// TwinCAT 3 PLC project WriteStringArrayToFile_Plc
// ProgramVersion: 3.1.4023.0
// libraries:
//   Tc2_Standard, * (Beckhoff Automation GmbH)
//   Tc2_System, * (Beckhoff Automation GmbH)
//   Tc3_Module, * (Beckhoff Automation GmbH)
// project tree:
//   / PlcTask.TcTTO
//   POUs/ FB_FillTestArray.TcPOU, FB_WriteStringArrayToFile.TcPOU, MAIN.TcPOU
// real-time tasks:
//   TASK PlcTask: cycle T#10ms, priority 20, ADS port 350

CONFIGURATION WriteStringArrayToFile_Plc
    RESOURCE PLC ON TwinCAT3
        TASK PlcTask(INTERVAL := T#10ms, PRIORITY := 20);
        PROGRAM MAIN WITH PlcTask : MAIN;
    END_RESOURCE
END_CONFIGURATION

// ---- POUs/MAIN.TcPOU
PROGRAM MAIN
VAR
	straTestStringArray	: ARRAY [1..10] OF STRING(255);
	fbFillArray	: FB_FillTestArray;
	fbWriteArray	: FB_WriteStringArrayToFile;
	
	bTestFillArray	: BOOL;
	bTestWriteArray	: BOOL;
	
	bTestOpen		: BOOL;
	bTestClose		: BOOL;
	
	fbFileOpen		: FB_FileOpen;
	fbFileClose		: FB_FileClose;
	
END_VAR

IF(_TaskInfo[GETCURTASKINDEXEX()].FirstCycle) THEN
	; // Do Nothing
END_IF


// Run the fill array FB 
fbFillArray(straArrayToFill	:= straTestStringArray);

// Run the file write array
fbWriteArray(straArrayToWrite	:= straTestStringArray);

IF(bTestFillArray) THEN
	fbFillArray.FillArray();
	bTestFillArray	:= FALSE;
END_IF

IF(bTestWriteArray) THEN
	fbWriteArray.WriteArray('C:\TestFile.txt');
	bTestWriteArray	:= FALSE;
END_IF

// Open the file - create it if it doesn't exist already
fbFileOpen(	sNetId 		:= '',
			sPathName 	:= 'C:\TestOpenFile.txt',
			nMode 		:= FOPEN_MODEAPPEND OR FOPEN_MODEPLUS,
			ePath 		:= PATH_GENERIC,
			bExecute 	:= bTestOpen,	
			tTimeout 	:= T#500MS);
			
// Close the file 
fbFileClose(sNetId :='' ,
			hFile := fbFileOpen.hFile,
			bExecute := fbFileOpen.hFile <> 0 AND bTestClose,
			tTimeout := T#500MS);

END_PROGRAM

// ---- POUs/FB_FillTestArray.TcPOU
FUNCTION_BLOCK FB_FillTestArray
VAR_IN_OUT
	straArrayToFill	: ARRAY[*] OF STRING(255);
END_VAR
VAR_INPUT
END_VAR
VAR_OUTPUT
END_VAR
VAR
	iIterator	: DINT;
END_VAR

METHOD FillArray : BOOL
VAR_INPUT
END_VAR
FOR iIterator:= LOWER_BOUND(straArrayToFill,1) TO UPPER_BOUND(straArrayToFill,1) BY 1 DO 
	straArrayToFill[iIterator]	:= CONCAT(CONCAT('Element Number : ',DINT_TO_STRING(iIterator)),'');
END_FOR
END_METHOD

END_FUNCTION_BLOCK

// ---- POUs/FB_WriteStringArrayToFile.TcPOU
FUNCTION_BLOCK FB_WriteStringArrayToFile
VAR_IN_OUT
	straArrayToWrite	: ARRAY[*] OF STRING(255);
END_VAR
VAR_OUTPUT
END_VAR
VAR
	
	fFallingFileOpenBusy 	: 	F_TRIG;	
	fFallingPutsBusy	 	:	F_TRIG;
	fFallingFileCloseBusy 	: 	F_TRIG;
	
	fbFileOpen 				: 	FB_FileOpen;
	fbFilePuts				: 	FB_FilePuts;
	fbFileClose 			: 	FB_FileClose;
	
	 
	strFilePath				: STRING(255);
	bTriggerWriteSequence	: BOOL;
	bRunFilePuts 			: BOOL;
	
	straStringArrayMirror	: ARRAY[1..1000] OF STRING(255);
	strStringToWrite		: STRING(255);
	
	diIterator		: DINT;
	diStringCount	: DINT;
	uiCurrentLine	: UINT	:= 1;
	
	uiStringPutsState	: UINT;
END_VAR

fFallingFileOpenBusy(CLK 	:= fbFileOpen.bBusy);
fFallingPutsBusy(	CLK 	:= fbFilePuts.bBusy);
fFallingFileCloseBusy(CLK	:= fbFileClose.bBusy); 

// Open the file - create it if it doesn't exist already
fbFileOpen(	sNetId 		:= '',
			sPathName 	:= strFilePath,
			nMode 		:= FOPEN_MODEAPPEND OR FOPEN_MODEPLUS,
			ePath 		:= PATH_GENERIC,
			bExecute 	:= bTriggerWriteSequence,	
			tTimeout 	:= T#500MS);

IF(bTriggerWriteSequence AND  fbFileOpen.hFile <> 0 AND fFallingFileOpenBusy.Q) THEN
	uiStringPutsState	:= 16#20;
END_IF

CASE uiStringPutsState OF 
	16#10:
		// Idle state
		uiCurrentLine	:= 1;
	
	16#20:	
		// trigger a line to be written
		bRunFilePuts		:= TRUE;	// trigger the write
		uiStringPutsState	:= 16#30;
	
	16#30:	
		// Increment the array index if there are more strings to be written
		
		bRunFilePuts	:= FALSE;
		
		IF fFallingPutsBusy.Q THEN
			
			IF(uiCurrentLine >= diStringCount) THEN
				uiStringPutsState	:= 16#10;
			ELSE
				uiCurrentLine		:= uiCurrentLine	+ 1;
				uiStringPutsState	:= 16#20;
			END_IF
			
		END_IF
			
	
	ELSE
;

END_CASE
		
// Write the current string to the file 	
fbFilePuts(	sNetId	:= '',
			hFile	:= fbFileOpen.hFile,
			sLine	:= straStringArrayMirror[uiCurrentLine],
			tTimeout	:= T#3000MS,
			bExecute	:= bRunFilePuts);

// Close the file 
fbFileClose(sNetId :='' ,
			hFile := fbFileOpen.hFile,
			bExecute := fbFileOpen.hFile <> 0 AND uiStringPutsState = 16#10,
			tTimeout := T#500MS);
		
// Reset the write sequence trigger when we are done closing the file
IF(fFallingFileCloseBusy.Q) THEN
	bTriggerWriteSequence	:= FALSE;
END_IF

METHOD AddCR : BOOL
VAR_INPUT
END_VAR
FOR diIterator	:= LOWER_BOUND(THIS^.straArrayToWrite,1) TO UPPER_BOUND(THIS^.straArrayToWrite,1) BY 1 DO 
	THIS^.straArrayToWrite[diIterator]	:= CONCAT(THIS^.straArrayToWrite[diIterator],'$0A');
END_FOR
END_METHOD

METHOD WriteArray : BOOL
VAR_INPUT
	strFilePath	: STRING(255);
END_VAR
THIS^.strFilePath	:= strFilePath;
THIS^.diStringCount	:= 0;

FOR diIterator:= LOWER_BOUND(THIS^.straArrayToWrite,1) TO UPPER_BOUND(THIS^.straArrayToWrite,1) BY 1 DO 
	THIS^.straStringArrayMirror[diIterator]	:= CONCAT(THIS^.straArrayToWrite[diIterator],'$0A');
	THIS^.diStringCount	:= THIS^.diStringCount	+ 1;
END_FOR

THIS^.bTriggerWriteSequence	:= TRUE;
END_METHOD

END_FUNCTION_BLOCK
